{region '#Template'}
	{attribute 'Version' := '1.2.2.0'}
	{attribute 'Tags' := '"LCID": "1031", "Text": "Universal, Valve"'}
	{attribute 'Tags' := '"LCID": "1033", "Text": "Universal, Valve"'}
	{attribute 'Using' := '"Type": "Template", "URI": "EC_AMEV"'}
	{attribute 'Using' := '"Type": "Template", "URI": "BA2_Param"'}
	{attribute 'Description' := '"LCID": "1031", "Text": "Ventil analog"'}
	{attribute 'Description' := '"LCID": "1033", "Text": "Valve analog"'}
{endregion}		 
FUNCTION_BLOCK FB_BA_Vlv EXTENDS FB_BA_ActuatorAnalog
VAR_INPUT
	bAblkLock				: BOOL;
END_VAR
VAR_OUTPUT
END_VAR
VAR_INPUT CONSTANT
	Ablk					: FB_BA_AntiBlocking;	
	Fdb						: FB_BA_AI_IO;		 
END_VAR

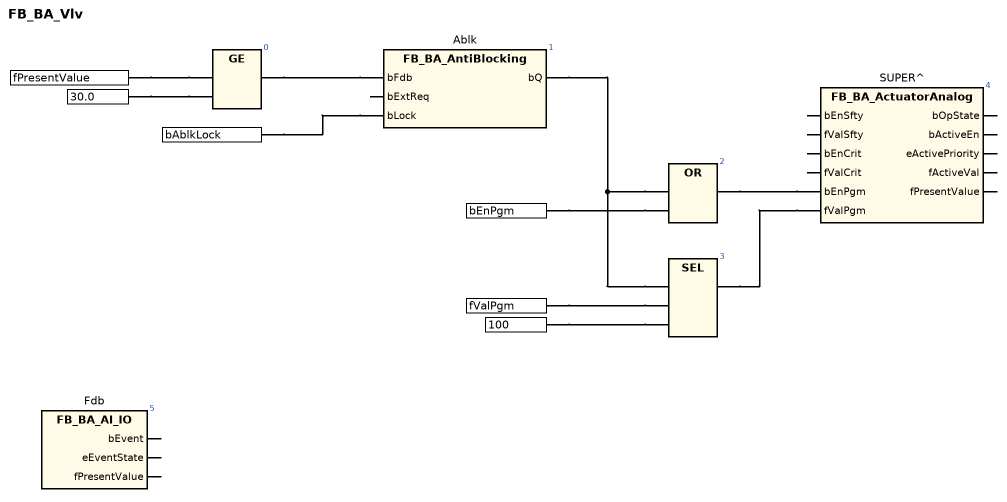
Ablk(bFdb := fPresentValue >= 30.0, bLock := bAblkLock); // FB_BA_AntiBlocking
SUPER^(bEnPgm := Ablk.bQ OR bEnPgm, fValPgm := SEL(Ablk.bQ, fValPgm, 100)); // FB_BA_ActuatorAnalog
Fdb(); // FB_BA_AI_IO

METHOD FB_init : BOOL
VAR_INPUT
	bInitRetains : BOOL; // if TRUE, the retain variables are initialized (warm start / cold start)
	bInCopyCode : BOOL;  // if TRUE, the instance afterwards gets moved into the copy code (online change)
END_VAR
Ablk.iParent					:= THIS^;	
Ablk.iLabel						:= LblUniFieldDevice.Valve_Ablk;
Ablk.sObjectName				:= '{Idx=01}';																	
Ablk.eDPADMode					:= E_BA_DPADMode.eIncludeDescription;	

Fdb.iParent						:= THIS^;		
Fdb.iLabel 						:= LblUniFieldDevice.Valve_Fdb;
Fdb.sObjectName					:= '{Idx=01}';
Fdb.sDeviceType					:= '';
Fdb.bEnOutOfService				:= FALSE;
Fdb.eUnit						:= E_BA_Unit.eOther_Percent;
Fdb.fResolution 				:= 0.03051851;
Fdb.fScaleOffset 				:= 0; 	
Fdb.fCOVIncrement				:= BA2_Param.fDefCOVIncrement;
Fdb.nEventClassID				:= EC_ID.NC80;
Fdb.stTimeDelay.nToNormal		:= BA2_Param.nDefTimeDelay_ToNormal;
Fdb.stTimeDelay.nToAbnormal		:= BA2_Param.nDefTimeDelay_ToAbnormal;
Fdb.stHighLimit.bEnable			:= FALSE;
Fdb.stHighLimit.fValue			:= 0.0;		
Fdb.stLowLimit.bEnable			:= FALSE;
Fdb.stLowLimit.fValue			:= 0.0;
Fdb.fLimitDeadband 				:= BA2_Param.fDefLimitDeadband;
Fdb.bAcknowledgeRm				:= FALSE;	
Fdb.aEventTransitionText[1]		:= txtEvent_Exceeded;
Fdb.aEventTransitionText[2]		:= txtEvent_Disturb;
Fdb.aEventTransitionText[3]		:= txtEvent_Normal;
Fdb.bEventDetectionEnable		:= FALSE;
Fdb.aEventEnable[1]				:= TRUE;			//	to_offnormal
Fdb.aEventEnable[2]				:= TRUE;			//	to_fault
Fdb.aEventEnable[3]				:= TRUE;			//	to_normal
Fdb.eEnPlantLock				:= E_BA_LockPriority.eNoLock;
END_METHOD

END_FUNCTION_BLOCK

(* stored: Version 1.1.0.1, ProductVersion 3.1.4024.9
   POU FB_BA_Vlv: Id {51eb23e0-0cbe-4d56-a096-aa87fdbfd250}, SpecialFunc None
   Method FB_init: Id {a2ce6982-f36d-48e0-92fd-30eb731612f6} *)
